{attribute 'linkalways'} 
{attribute 'no_explicit_call' := 'This FB is a CLASS and must be accessed using methods or properties'}
{attribute 'enable_dynamic_creation'}
FUNCTION_BLOCK _ETcVnSolvePnPMethod EXTENDS EnumDatatypeBase
VAR
	localData : ETcVnSolvePnPMethod;
	activeData : REFERENCE TO ETcVnSolvePnPMethod;
	enumBaseDatatype : _DINT(localData);
END_VAR

METHOD PRIVATE AddLocalEnumeration
VAR_INPUT
	Enumeration : T_MAXSTRING;
	Value : ETcVnSolvePnPMethod;
END_VAR
AddEnumeration(Enumeration, Value);
END_METHOD

PROPERTY PUBLIC Address : PVOID
GET
Address := ADR(activeData);
END_GET
END_PROPERTY

METHOD PUBLIC ClearReference
VAR_INPUT
END_VAR
activeData REF= localData;
SetBaseDatatypeReference();
END_METHOD

METHOD PUBLIC Clone : I_Datatype
VAR
    pClone : POINTER TO _ETcVnSolvePnPMethod;
END_VAR
pClone := __NEW(_ETcVnSolvePnPMethod(InitialValue := Value));
Clone := pClone^;
END_METHOD

METHOD FB_init : BOOL
VAR_INPUT
	bInitRetains : BOOL; // if TRUE, the retain variables are initialized (warm start / cold start)
	bInCopyCode : BOOL;  // if TRUE, the instance afterwards gets moved into the copy code (online change)
	InitialValue : ETcVnSolvePnPMethod;
END_VAR
localData := InitialValue;
AddBaseDatatype(enumBaseDatatype);
ClearReference();

AddLocalEnumeration('TCVN_SPM_ITERATIVE', ETcVnSolvePnPMethod.TCVN_SPM_ITERATIVE);
AddLocalEnumeration('TCVN_SPM_EPNP', ETcVnSolvePnPMethod.TCVN_SPM_EPNP);
AddLocalEnumeration('TCVN_SPM_P3P', ETcVnSolvePnPMethod.TCVN_SPM_P3P);
AddLocalEnumeration('TCVN_SPM_AP3P', ETcVnSolvePnPMethod.TCVN_SPM_AP3P);
AddLocalEnumeration('TCVN_SPM_IPPE', ETcVnSolvePnPMethod.TCVN_SPM_IPPE);
AddLocalEnumeration('TCVN_SPM_IPPE_SQUARE', ETcVnSolvePnPMethod.TCVN_SPM_IPPE_SQUARE);
AddLocalEnumeration('TCVN_SPM_SQPNP', ETcVnSolvePnPMethod.TCVN_SPM_SQPNP);
END_METHOD

PROPERTY PUBLIC Identifier : T_MAXSTRING
GET
Identifier := 'ETcVnSolvePnPMethod';
END_GET
END_PROPERTY

METHOD IsEnumeratorValueEqual : BOOL
VAR_INPUT
	Enumerator : I_KeyValueForwardEnumerator;
END_VAR
VAR
	storedValue : ETcVnSolvePnPMethod;
END_VAR
IF NOT Enumerator.TryGet(storedValue) THEN
	RETURN;
END_IF

IsEnumeratorValueEqual := storedValue = activeData;
END_METHOD

METHOD PUBLIC MakeReferenceTo
VAR_INPUT
	ReferenceTarget : REFERENCE TO ETcVnSolvePnPMethod;
END_VAR
activeData REF= ReferenceTarget;
SetBaseDatatypeReference();
END_METHOD

METHOD PROTECTED SetBaseDatatypeReference
VAR_INPUT
END_VAR
enumBaseDatatype.MakeReferenceTo(activeData);
END_METHOD

PROPERTY PUBLIC Size : UDINT
GET
Size := SIZEOF(activeData);
END_GET
END_PROPERTY

METHOD TryMakeReferenceTo : BOOL
VAR_INPUT
	Target : I_Datatype;
END_VAR
VAR
	targetAsEnum : I_EnumDatatype;
	pTargetData : POINTER TO ETcVnSolvePnPMethod;
END_VAR
IF NOT Target.TryResolveAsEnumDatatype(targetAsEnum) THEN
	RETURN;
END_IF

IF targetAsEnum.Identifier <> Identifier THEN
	RETURN;
END_IF

pTargetData := Target.Address;
activeData REF= pTargetData^;
SetBaseDatatypeReference();
TryMakeReferenceTo := TRUE;
END_METHOD

PROPERTY PUBLIC Value : ETcVnSolvePnPMethod
GET
Value := activeData;
END_GET
SET
activeData := Value;
END_SET
END_PROPERTY

END_FUNCTION_BLOCK

(* stored: Version 1.1.0.1, ProductVersion 3.1.4024.12
   POU _ETcVnSolvePnPMethod: Id {93e8093c-f0d3-0ae1-1c04-9acab1a62f3b}, SpecialFunc None
   Folder Constructor: Id {e1e72cd6-2121-0341-3a12-482c02a9bec6}
   Folder Private: Id {0d7004be-713a-016e-12e9-06370cbd39a0}
   Folder Protected: Id {a9b2e5fb-7f96-04e7-2b6e-2ec8fcc537cf}
   Method AddLocalEnumeration: Id {7189cee1-cf8c-0819-1788-41e6672bbdfa}
   Property Address: Id {9c426067-a701-0a1a-0006-819d66754aa1}
   Get Get: Id {b5683506-0b6a-07e8-12d7-431c58a17eaf}
   Method ClearReference: Id {788c60e4-eae7-007a-31a1-4989083beb19}
   Method Clone: Id {321b22b2-fd82-0fa7-2ed0-d75bb22d13d4}
   Method FB_init: Id {1bbb8533-c197-0d09-0b73-b8470fea1c8c}
   Property Identifier: Id {4a34e66d-68ec-0440-31bb-73f0b169bf20}
   Get Get: Id {740fbe4c-3d47-0c4a-03ba-938b2dcef0af}
   Method IsEnumeratorValueEqual: Id {e3e44a9e-0bec-09b5-212b-09a2c1514c5f}
   Method MakeReferenceTo: Id {42533c2a-89a9-09ce-08a5-4b97ea228537}
   Method SetBaseDatatypeReference: Id {fe208d05-a832-0922-2237-d55088fd5abe}
   Property Size: Id {3b550fed-c3c2-030f-3c8f-b4c764f827b8}
   Get Get: Id {e9c5aada-9166-001e-1e03-dd4073d2eb8e}
   Method TryMakeReferenceTo: Id {4ac1763b-39ce-0726-26fc-510432fb6ccc}
   Property Value: Id {258044b2-c23a-0509-2688-7c17eac4834c}
   Get Get: Id {229e6db7-a840-0490-19c5-33246ca5e40e}
   Set Set: Id {f7440bb4-bec9-0b62-3002-3881b70c97ad} *)
